# EPICS autosave request: iocBoot/iocLinux/auto_settings.req
file built_settings.req P=$(P)
file DCMotorServer.req P=$(P)dcm:
